INTERFACE I_Nodes

METHOD PUBLIC Accept
VAR_INPUT
	Visitor : I_NodeVisitor;
END_VAR
END_METHOD

METHOD AddNode
VAR_INPUT
	Node : I_Node;
END_VAR
END_METHOD

METHOD PUBLIC GetNodesInOrderEnumerator : I_ForwardEnumerator
VAR_INPUT
END_VAR
END_METHOD

PROPERTY PUBLIC HasNodes : BOOL
GET
END_GET
END_PROPERTY

METHOD PUBLIC TryGetNodeById : BOOL
VAR_INPUT
	Id : T_MAXSTRING;
	Destination : REFERENCE TO I_Node;
END_VAR
END_METHOD

END_INTERFACE

(* stored: Version 1.1.0.1, ProductVersion 3.1.4024.13
   Itf I_Nodes: Id {c7bb15f9-1eb4-436a-9915-c62c2fbf6d53}
   Method Accept: Id {075c2acf-8b17-488d-9dc7-c94280aab56d}
   Method AddNode: Id {7c6ef1cb-77dd-4b7a-b9b8-e23e3e7b0e99}
   Method GetNodesInOrderEnumerator: Id {a531acc3-9a79-0d0c-28ea-eb9a4f88d6dc}
   Property HasNodes: Id {608d2b7e-39ad-04a0-20b2-169ee296276d}
   Get Get: Id {c8564dc9-675b-0ae6-116c-1a5e907b6ea7}
   Method TryGetNodeById: Id {08a8932c-41d1-49f6-947f-fc49e0d12e42} *)
